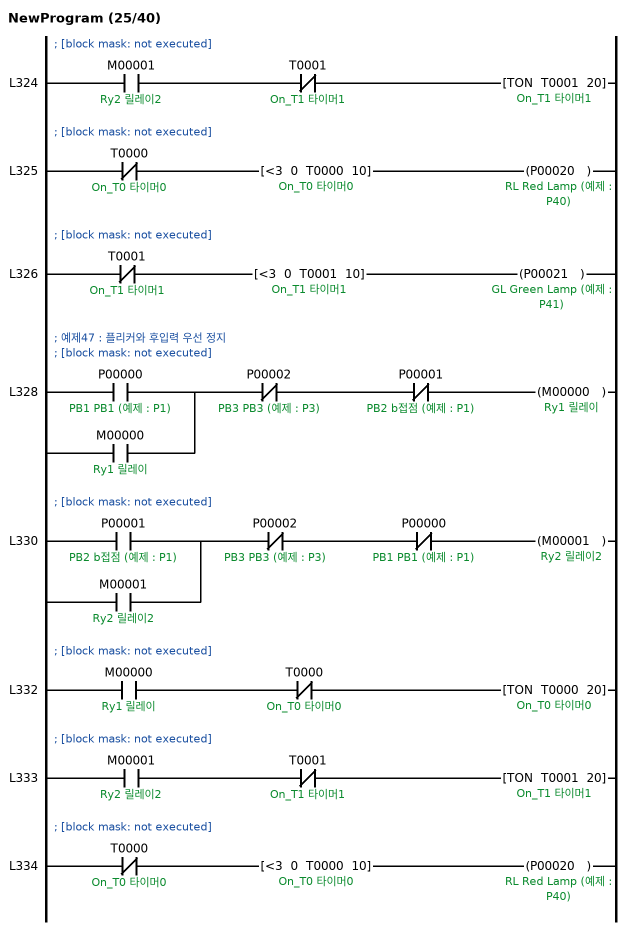
[picture p24: NewProgram rungs L324-L334]
; L324 (block mask: not executed)
LOAD      M00001	// Ry2 릴레이2
AND NOT   T0001	// On_T1 타이머1
TON       T0001 20	// On_T1 타이머1
; L325 (block mask: not executed)
LOAD NOT  T0000	// On_T0 타이머0
AND<3     0 T0000 10	// On_T0 타이머0
OUT       P00020	// RL Red Lamp (예제 : P40)
; L326 (block mask: not executed)
LOAD NOT  T0001	// On_T1 타이머1
AND<3     0 T0001 10	// On_T1 타이머1
OUT       P00021	// GL Green Lamp (예제 : P41)
// 예제47 : 플리커와 후입력 우선 정지
; L328 (block mask: not executed)
LOAD      P00000	// PB1 PB1 (예제 : P1)
OR        M00000	// Ry1 릴레이
AND NOT   P00002	// PB3 PB3 (예제 : P3)
AND NOT   P00001	// PB2 b접점 (예제 : P1)
OUT       M00000	// Ry1 릴레이
; L330 (block mask: not executed)
LOAD      P00001	// PB2 b접점 (예제 : P1)
OR        M00001	// Ry2 릴레이2
AND NOT   P00002	// PB3 PB3 (예제 : P3)
AND NOT   P00000	// PB1 PB1 (예제 : P1)
OUT       M00001	// Ry2 릴레이2
; L332 (block mask: not executed)
LOAD      M00000	// Ry1 릴레이
AND NOT   T0000	// On_T0 타이머0
TON       T0000 20	// On_T0 타이머0
; L333 (block mask: not executed)
LOAD      M00001	// Ry2 릴레이2
AND NOT   T0001	// On_T1 타이머1
TON       T0001 20	// On_T1 타이머1
; L334 (block mask: not executed)
LOAD NOT  T0000	// On_T0 타이머0
AND<3     0 T0000 10	// On_T0 타이머0
OUT       P00020	// RL Red Lamp (예제 : P40)

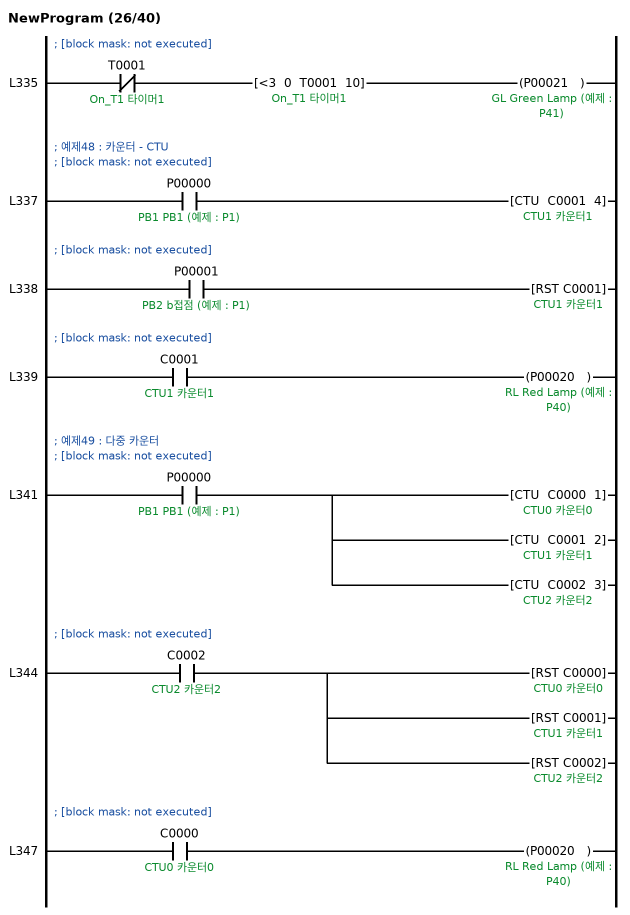
; L335 (block mask: not executed)
LOAD NOT  T0001	// On_T1 타이머1
AND<3     0 T0001 10	// On_T1 타이머1
OUT       P00021	// GL Green Lamp (예제 : P41)
// 예제48 : 카운터 - CTU
; L337 (block mask: not executed)
LOAD      P00000	// PB1 PB1 (예제 : P1)
CTU       C0001 4	// CTU1 카운터1
; L338 (block mask: not executed)
LOAD      P00001	// PB2 b접점 (예제 : P1)
RST       C0001	// CTU1 카운터1
; L339 (block mask: not executed)
LOAD      C0001	// CTU1 카운터1
OUT       P00020	// RL Red Lamp (예제 : P40)
// 예제49 : 다중 카운터
; L341 (block mask: not executed)
LOAD      P00000	// PB1 PB1 (예제 : P1)
CTU       C0000 1	// CTU0 카운터0
CTU       C0001 2	// CTU1 카운터1
CTU       C0002 3	// CTU2 카운터2
; L344 (block mask: not executed)
LOAD      C0002	// CTU2 카운터2
RST       C0000	// CTU0 카운터0
RST       C0001	// CTU1 카운터1
RST       C0002	// CTU2 카운터2
; L347 (block mask: not executed)
LOAD      C0000	// CTU0 카운터0
OUT       P00020	// RL Red Lamp (예제 : P40)

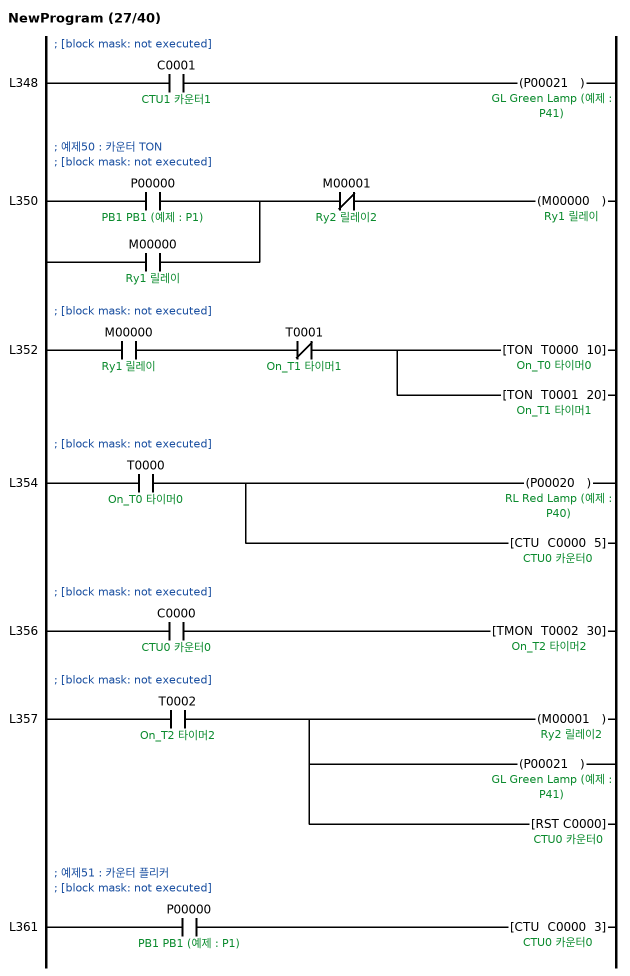
; L348 (block mask: not executed)
LOAD      C0001	// CTU1 카운터1
OUT       P00021	// GL Green Lamp (예제 : P41)
// 예제50 : 카운터 TON
; L350 (block mask: not executed)
LOAD      P00000	// PB1 PB1 (예제 : P1)
OR        M00000	// Ry1 릴레이
AND NOT   M00001	// Ry2 릴레이2
OUT       M00000	// Ry1 릴레이
; L352 (block mask: not executed)
LOAD      M00000	// Ry1 릴레이
AND NOT   T0001	// On_T1 타이머1
TON       T0000 10	// On_T0 타이머0
TON       T0001 20	// On_T1 타이머1
; L354 (block mask: not executed)
LOAD      T0000	// On_T0 타이머0
OUT       P00020	// RL Red Lamp (예제 : P40)
CTU       C0000 5	// CTU0 카운터0
; L356 (block mask: not executed)
LOAD      C0000	// CTU0 카운터0
TMON      T0002 30	// On_T2 타이머2
; L357 (block mask: not executed)
LOAD      T0002	// On_T2 타이머2
OUT       M00001	// Ry2 릴레이2
OUT       P00021	// GL Green Lamp (예제 : P41)
RST       C0000	// CTU0 카운터0
// 예제51 : 카운터 플리커
; L361 (block mask: not executed)
LOAD      P00000	// PB1 PB1 (예제 : P1)
CTU       C0000 3	// CTU0 카운터0

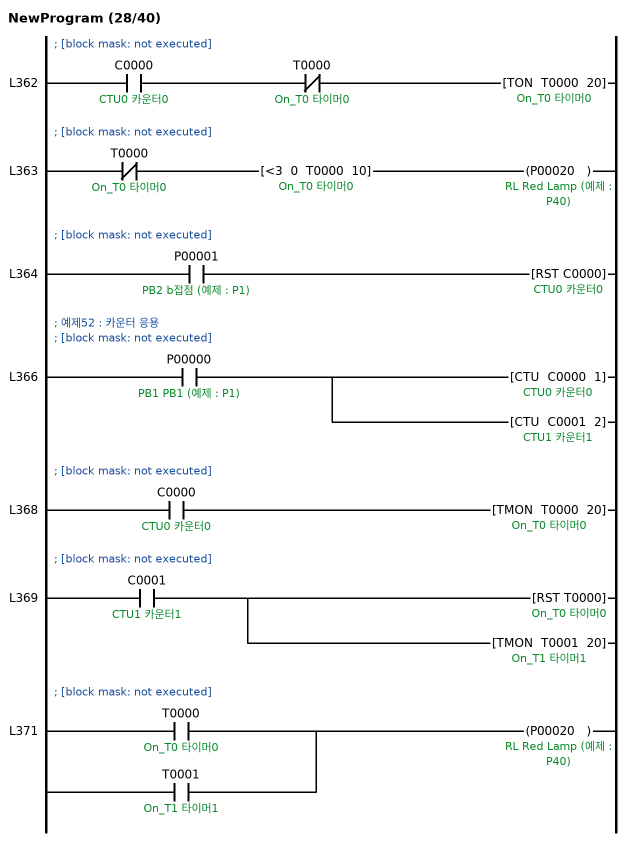
; L362 (block mask: not executed)
LOAD      C0000	// CTU0 카운터0
AND NOT   T0000	// On_T0 타이머0
TON       T0000 20	// On_T0 타이머0
; L363 (block mask: not executed)
LOAD NOT  T0000	// On_T0 타이머0
AND<3     0 T0000 10	// On_T0 타이머0
OUT       P00020	// RL Red Lamp (예제 : P40)
; L364 (block mask: not executed)
LOAD      P00001	// PB2 b접점 (예제 : P1)
RST       C0000	// CTU0 카운터0
// 예제52 : 카운터 응용
; L366 (block mask: not executed)
LOAD      P00000	// PB1 PB1 (예제 : P1)
CTU       C0000 1	// CTU0 카운터0
CTU       C0001 2	// CTU1 카운터1
; L368 (block mask: not executed)
LOAD      C0000	// CTU0 카운터0
TMON      T0000 20	// On_T0 타이머0
; L369 (block mask: not executed)
LOAD      C0001	// CTU1 카운터1
RST       T0000	// On_T0 타이머0
TMON      T0001 20	// On_T1 타이머1
; L371 (block mask: not executed)
LOAD      T0000	// On_T0 타이머0
OR        T0001	// On_T1 타이머1
OUT       P00020	// RL Red Lamp (예제 : P40)

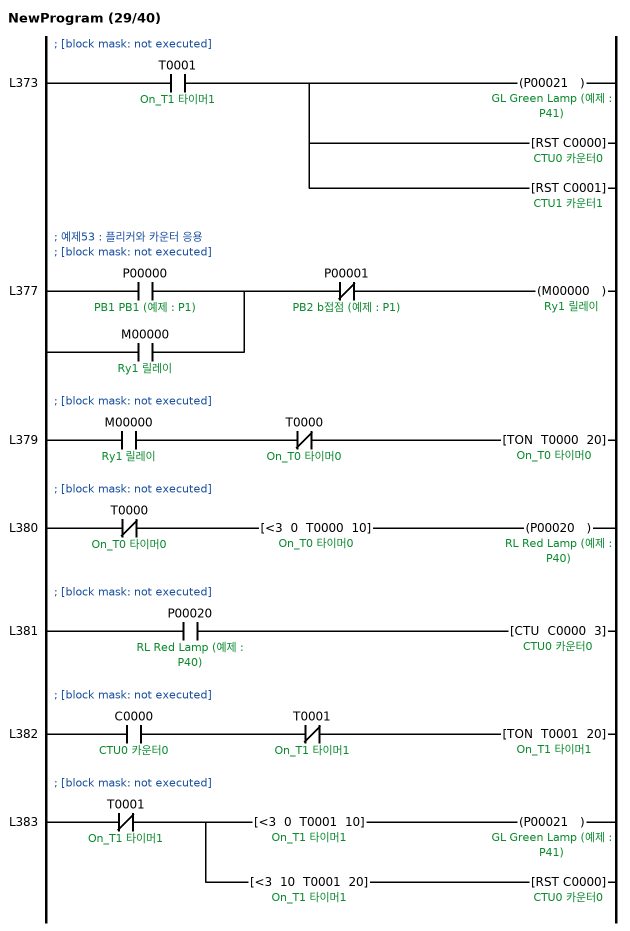
; L373 (block mask: not executed)
LOAD      T0001	// On_T1 타이머1
OUT       P00021	// GL Green Lamp (예제 : P41)
RST       C0000	// CTU0 카운터0
RST       C0001	// CTU1 카운터1
// 예제53 : 플리커와 카운터 응용
; L377 (block mask: not executed)
LOAD      P00000	// PB1 PB1 (예제 : P1)
OR        M00000	// Ry1 릴레이
AND NOT   P00001	// PB2 b접점 (예제 : P1)
OUT       M00000	// Ry1 릴레이
; L379 (block mask: not executed)
LOAD      M00000	// Ry1 릴레이
AND NOT   T0000	// On_T0 타이머0
TON       T0000 20	// On_T0 타이머0
; L380 (block mask: not executed)
LOAD NOT  T0000	// On_T0 타이머0
AND<3     0 T0000 10	// On_T0 타이머0
OUT       P00020	// RL Red Lamp (예제 : P40)
; L381 (block mask: not executed)
LOAD      P00020	// RL Red Lamp (예제 : P40)
CTU       C0000 3	// CTU0 카운터0
; L382 (block mask: not executed)
LOAD      C0000	// CTU0 카운터0
AND NOT   T0001	// On_T1 타이머1
TON       T0001 20	// On_T1 타이머1
; L383 (block mask: not executed)
LOAD NOT  T0001	// On_T1 타이머1
MPUSH
AND<3     0 T0001 10	// On_T1 타이머1
OUT       P00021	// GL Green Lamp (예제 : P41)
MPOP
AND<3     10 T0001 20	// On_T1 타이머1
RST       C0000	// CTU0 카운터0

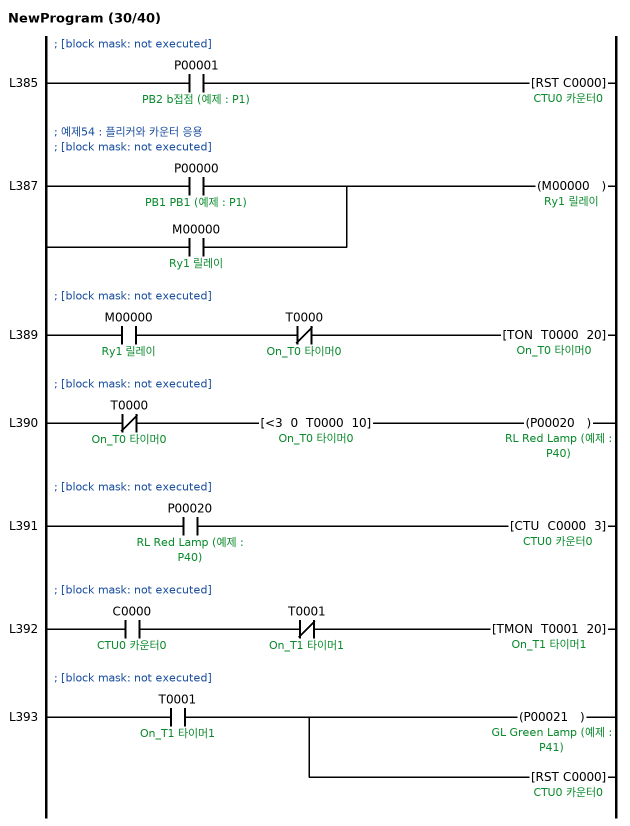
; L385 (block mask: not executed)
LOAD      P00001	// PB2 b접점 (예제 : P1)
RST       C0000	// CTU0 카운터0
// 예제54 : 플리커와 카운터 응용
; L387 (block mask: not executed)
LOAD      P00000	// PB1 PB1 (예제 : P1)
OR        M00000	// Ry1 릴레이
OUT       M00000	// Ry1 릴레이
; L389 (block mask: not executed)
LOAD      M00000	// Ry1 릴레이
AND NOT   T0000	// On_T0 타이머0
TON       T0000 20	// On_T0 타이머0
; L390 (block mask: not executed)
LOAD NOT  T0000	// On_T0 타이머0
AND<3     0 T0000 10	// On_T0 타이머0
OUT       P00020	// RL Red Lamp (예제 : P40)
; L391 (block mask: not executed)
LOAD      P00020	// RL Red Lamp (예제 : P40)
CTU       C0000 3	// CTU0 카운터0
; L392 (block mask: not executed)
LOAD      C0000	// CTU0 카운터0
AND NOT   T0001	// On_T1 타이머1
TMON      T0001 20	// On_T1 타이머1
; L393 (block mask: not executed)
LOAD      T0001	// On_T1 타이머1
OUT       P00021	// GL Green Lamp (예제 : P41)
RST       C0000	// CTU0 카운터0

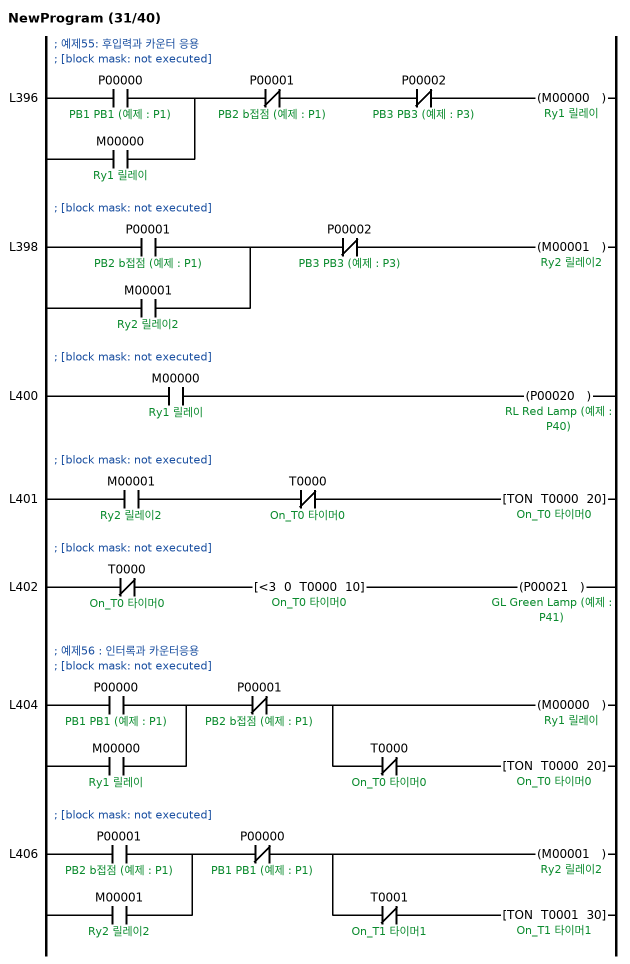
// 예제55: 후입력과 카운터 응용
; L396 (block mask: not executed)
LOAD      P00000	// PB1 PB1 (예제 : P1)
OR        M00000	// Ry1 릴레이
AND NOT   P00001	// PB2 b접점 (예제 : P1)
AND NOT   P00002	// PB3 PB3 (예제 : P3)
OUT       M00000	// Ry1 릴레이
; L398 (block mask: not executed)
LOAD      P00001	// PB2 b접점 (예제 : P1)
OR        M00001	// Ry2 릴레이2
AND NOT   P00002	// PB3 PB3 (예제 : P3)
OUT       M00001	// Ry2 릴레이2
; L400 (block mask: not executed)
LOAD      M00000	// Ry1 릴레이
OUT       P00020	// RL Red Lamp (예제 : P40)
; L401 (block mask: not executed)
LOAD      M00001	// Ry2 릴레이2
AND NOT   T0000	// On_T0 타이머0
TON       T0000 20	// On_T0 타이머0
; L402 (block mask: not executed)
LOAD NOT  T0000	// On_T0 타이머0
AND<3     0 T0000 10	// On_T0 타이머0
OUT       P00021	// GL Green Lamp (예제 : P41)
// 예제56 : 인터록과 카운터응용
; L404 (block mask: not executed)
LOAD      P00000	// PB1 PB1 (예제 : P1)
OR        M00000	// Ry1 릴레이
AND NOT   P00001	// PB2 b접점 (예제 : P1)
OUT       M00000	// Ry1 릴레이
AND NOT   T0000	// On_T0 타이머0
TON       T0000 20	// On_T0 타이머0
; L406 (block mask: not executed)
LOAD      P00001	// PB2 b접점 (예제 : P1)
OR        M00001	// Ry2 릴레이2
AND NOT   P00000	// PB1 PB1 (예제 : P1)
OUT       M00001	// Ry2 릴레이2
AND NOT   T0001	// On_T1 타이머1
TON       T0001 30	// On_T1 타이머1

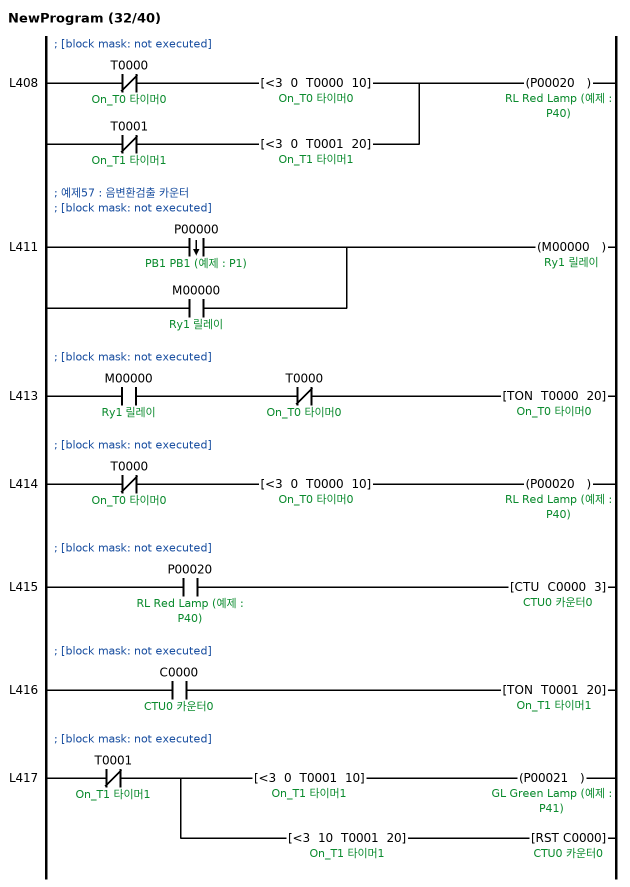
; L408 (block mask: not executed)
LOAD NOT  T0000	// On_T0 타이머0
AND<3     0 T0000 10	// On_T0 타이머0
LOAD NOT  T0001	// On_T1 타이머1
AND<3     0 T0001 20	// On_T1 타이머1
OR LOAD
OUT       P00020	// RL Red Lamp (예제 : P40)
// 예제57 : 음변환검출 카운터
; L411 (block mask: not executed)
LOADN     P00000	// PB1 PB1 (예제 : P1)
OR        M00000	// Ry1 릴레이
OUT       M00000	// Ry1 릴레이
; L413 (block mask: not executed)
LOAD      M00000	// Ry1 릴레이
AND NOT   T0000	// On_T0 타이머0
TON       T0000 20	// On_T0 타이머0
; L414 (block mask: not executed)
LOAD NOT  T0000	// On_T0 타이머0
AND<3     0 T0000 10	// On_T0 타이머0
OUT       P00020	// RL Red Lamp (예제 : P40)
; L415 (block mask: not executed)
LOAD      P00020	// RL Red Lamp (예제 : P40)
CTU       C0000 3	// CTU0 카운터0
; L416 (block mask: not executed)
LOAD      C0000	// CTU0 카운터0
TON       T0001 20	// On_T1 타이머1
; L417 (block mask: not executed)
LOAD NOT  T0001	// On_T1 타이머1
MPUSH
AND<3     0 T0001 10	// On_T1 타이머1
OUT       P00021	// GL Green Lamp (예제 : P41)
MPOP
AND<3     10 T0001 20	// On_T1 타이머1
RST       C0000	// CTU0 카운터0

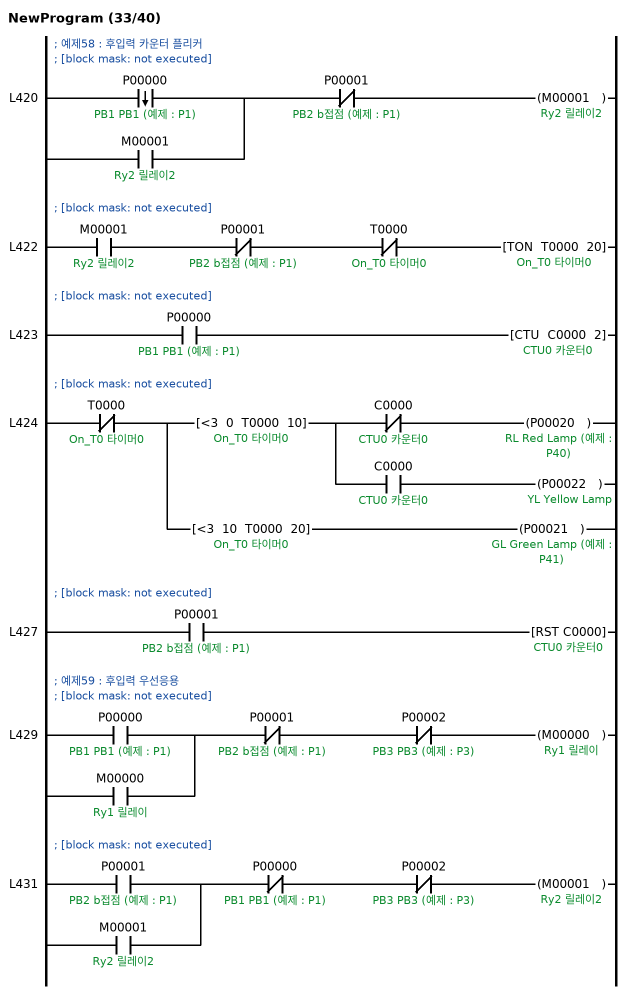
// 예제58 : 후입력 카운터 플리커
; L420 (block mask: not executed)
LOADN     P00000	// PB1 PB1 (예제 : P1)
OR        M00001	// Ry2 릴레이2
AND NOT   P00001	// PB2 b접점 (예제 : P1)
OUT       M00001	// Ry2 릴레이2
; L422 (block mask: not executed)
LOAD      M00001	// Ry2 릴레이2
AND NOT   P00001	// PB2 b접점 (예제 : P1)
AND NOT   T0000	// On_T0 타이머0
TON       T0000 20	// On_T0 타이머0
; L423 (block mask: not executed)
LOAD      P00000	// PB1 PB1 (예제 : P1)
CTU       C0000 2	// CTU0 카운터0
; L424 (block mask: not executed)
LOAD NOT  T0000	// On_T0 타이머0
MPUSH
AND<3     0 T0000 10	// On_T0 타이머0
MPUSH
AND NOT   C0000	// CTU0 카운터0
OUT       P00020	// RL Red Lamp (예제 : P40)
MPOP
AND       C0000	// CTU0 카운터0
OUT       P00022	// YL Yellow Lamp
MPOP
AND<3     10 T0000 20	// On_T0 타이머0
OUT       P00021	// GL Green Lamp (예제 : P41)
; L427 (block mask: not executed)
LOAD      P00001	// PB2 b접점 (예제 : P1)
RST       C0000	// CTU0 카운터0
// 예제59 : 후입력 우선응용
; L429 (block mask: not executed)
LOAD      P00000	// PB1 PB1 (예제 : P1)
OR        M00000	// Ry1 릴레이
AND NOT   P00001	// PB2 b접점 (예제 : P1)
AND NOT   P00002	// PB3 PB3 (예제 : P3)
OUT       M00000	// Ry1 릴레이
; L431 (block mask: not executed)
LOAD      P00001	// PB2 b접점 (예제 : P1)
OR        M00001	// Ry2 릴레이2
AND NOT   P00000	// PB1 PB1 (예제 : P1)
AND NOT   P00002	// PB3 PB3 (예제 : P3)
OUT       M00001	// Ry2 릴레이2

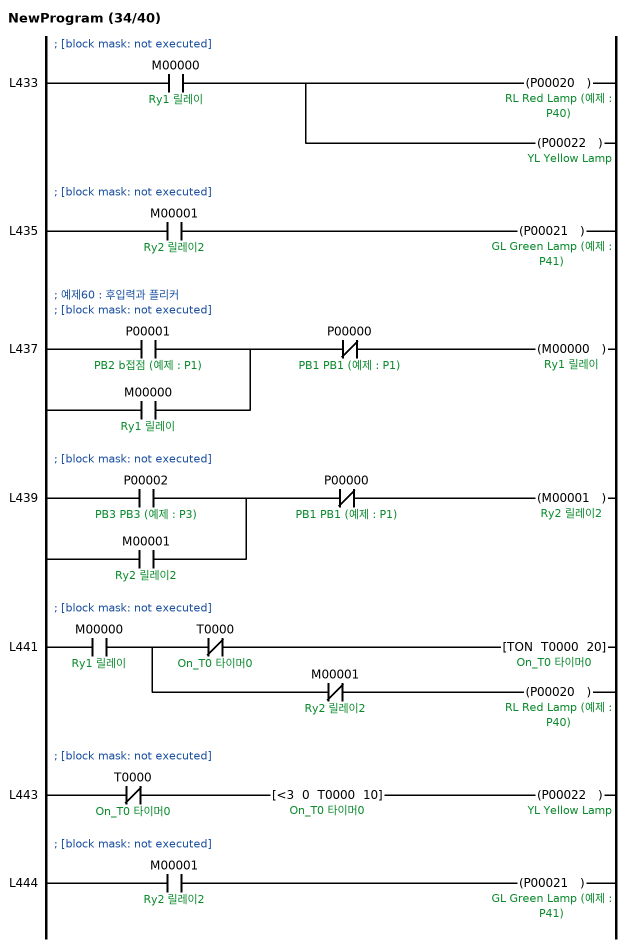
; L433 (block mask: not executed)
LOAD      M00000	// Ry1 릴레이
OUT       P00020	// RL Red Lamp (예제 : P40)
OUT       P00022	// YL Yellow Lamp
; L435 (block mask: not executed)
LOAD      M00001	// Ry2 릴레이2
OUT       P00021	// GL Green Lamp (예제 : P41)
// 예제60 : 후입력과 플리커
; L437 (block mask: not executed)
LOAD      P00001	// PB2 b접점 (예제 : P1)
OR        M00000	// Ry1 릴레이
AND NOT   P00000	// PB1 PB1 (예제 : P1)
OUT       M00000	// Ry1 릴레이
; L439 (block mask: not executed)
LOAD      P00002	// PB3 PB3 (예제 : P3)
OR        M00001	// Ry2 릴레이2
AND NOT   P00000	// PB1 PB1 (예제 : P1)
OUT       M00001	// Ry2 릴레이2
; L441 (block mask: not executed)
LOAD      M00000	// Ry1 릴레이
MPUSH
AND NOT   T0000	// On_T0 타이머0
TON       T0000 20	// On_T0 타이머0
MPOP
AND NOT   M00001	// Ry2 릴레이2
OUT       P00020	// RL Red Lamp (예제 : P40)
; L443 (block mask: not executed)
LOAD NOT  T0000	// On_T0 타이머0
AND<3     0 T0000 10	// On_T0 타이머0
OUT       P00022	// YL Yellow Lamp
; L444 (block mask: not executed)
LOAD      M00001	// Ry2 릴레이2
OUT       P00021	// GL Green Lamp (예제 : P41)

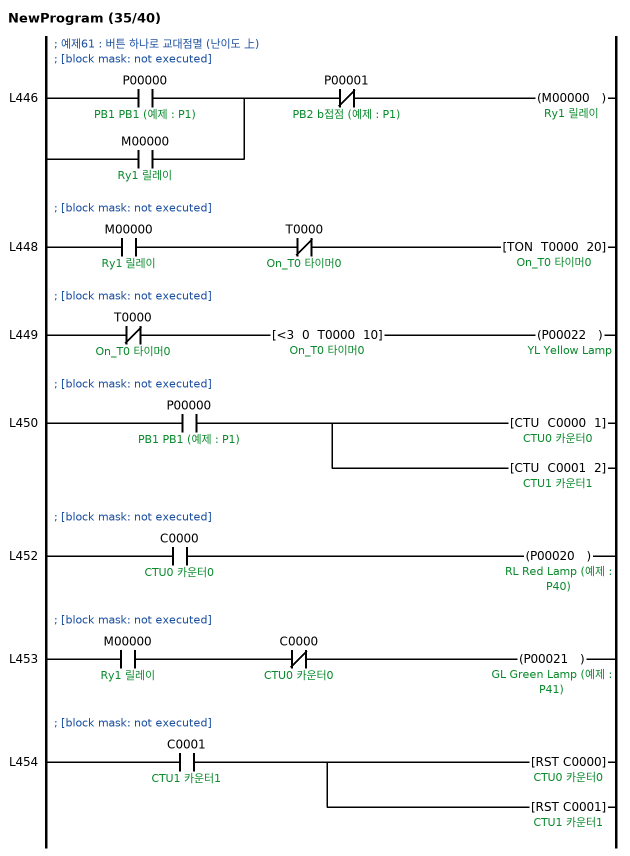
// 예제61 : 버튼 하나로 교대점멸 (난이도 上)
; L446 (block mask: not executed)
LOAD      P00000	// PB1 PB1 (예제 : P1)
OR        M00000	// Ry1 릴레이
AND NOT   P00001	// PB2 b접점 (예제 : P1)
OUT       M00000	// Ry1 릴레이
; L448 (block mask: not executed)
LOAD      M00000	// Ry1 릴레이
AND NOT   T0000	// On_T0 타이머0
TON       T0000 20	// On_T0 타이머0
; L449 (block mask: not executed)
LOAD NOT  T0000	// On_T0 타이머0
AND<3     0 T0000 10	// On_T0 타이머0
OUT       P00022	// YL Yellow Lamp
; L450 (block mask: not executed)
LOAD      P00000	// PB1 PB1 (예제 : P1)
CTU       C0000 1	// CTU0 카운터0
CTU       C0001 2	// CTU1 카운터1
; L452 (block mask: not executed)
LOAD      C0000	// CTU0 카운터0
OUT       P00020	// RL Red Lamp (예제 : P40)
; L453 (block mask: not executed)
LOAD      M00000	// Ry1 릴레이
AND NOT   C0000	// CTU0 카운터0
OUT       P00021	// GL Green Lamp (예제 : P41)
; L454 (block mask: not executed)
LOAD      C0001	// CTU1 카운터1
RST       C0000	// CTU0 카운터0
RST       C0001	// CTU1 카운터1

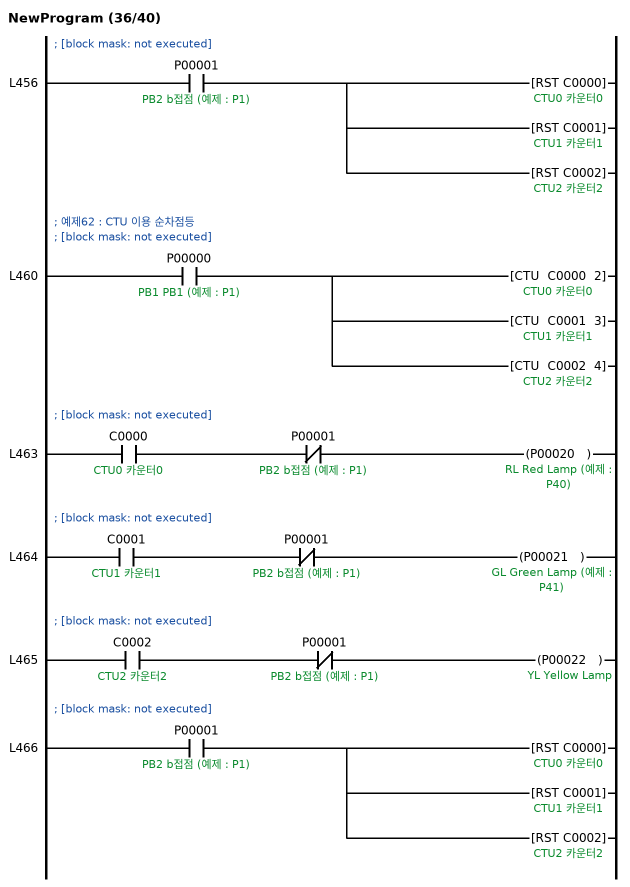
; L456 (block mask: not executed)
LOAD      P00001	// PB2 b접점 (예제 : P1)
RST       C0000	// CTU0 카운터0
RST       C0001	// CTU1 카운터1
RST       C0002	// CTU2 카운터2
// 예제62 : CTU 이용 순차점등
; L460 (block mask: not executed)
LOAD      P00000	// PB1 PB1 (예제 : P1)
CTU       C0000 2	// CTU0 카운터0
CTU       C0001 3	// CTU1 카운터1
CTU       C0002 4	// CTU2 카운터2
; L463 (block mask: not executed)
LOAD      C0000	// CTU0 카운터0
AND NOT   P00001	// PB2 b접점 (예제 : P1)
OUT       P00020	// RL Red Lamp (예제 : P40)
; L464 (block mask: not executed)
LOAD      C0001	// CTU1 카운터1
AND NOT   P00001	// PB2 b접점 (예제 : P1)
OUT       P00021	// GL Green Lamp (예제 : P41)
; L465 (block mask: not executed)
LOAD      C0002	// CTU2 카운터2
AND NOT   P00001	// PB2 b접점 (예제 : P1)
OUT       P00022	// YL Yellow Lamp
; L466 (block mask: not executed)
LOAD      P00001	// PB2 b접점 (예제 : P1)
RST       C0000	// CTU0 카운터0
RST       C0001	// CTU1 카운터1
RST       C0002	// CTU2 카운터2

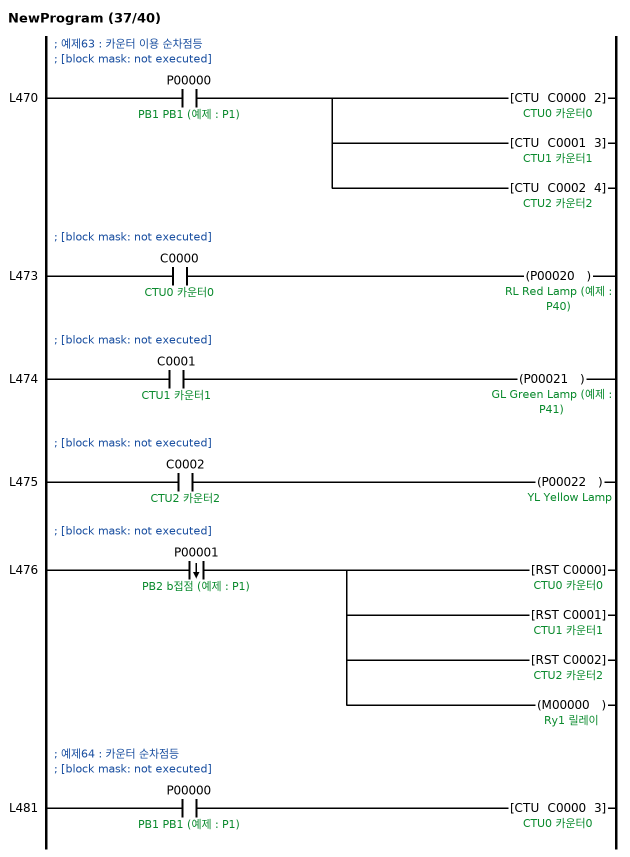
// 예제63 : 카운터 이용 순차점등
; L470 (block mask: not executed)
LOAD      P00000	// PB1 PB1 (예제 : P1)
CTU       C0000 2	// CTU0 카운터0
CTU       C0001 3	// CTU1 카운터1
CTU       C0002 4	// CTU2 카운터2
; L473 (block mask: not executed)
LOAD      C0000	// CTU0 카운터0
OUT       P00020	// RL Red Lamp (예제 : P40)
; L474 (block mask: not executed)
LOAD      C0001	// CTU1 카운터1
OUT       P00021	// GL Green Lamp (예제 : P41)
; L475 (block mask: not executed)
LOAD      C0002	// CTU2 카운터2
OUT       P00022	// YL Yellow Lamp
; L476 (block mask: not executed)
LOADN     P00001	// PB2 b접점 (예제 : P1)
RST       C0000	// CTU0 카운터0
RST       C0001	// CTU1 카운터1
RST       C0002	// CTU2 카운터2
OUT       M00000	// Ry1 릴레이
// 예제64 : 카운터 순차점등
; L481 (block mask: not executed)
LOAD      P00000	// PB1 PB1 (예제 : P1)
CTU       C0000 3	// CTU0 카운터0

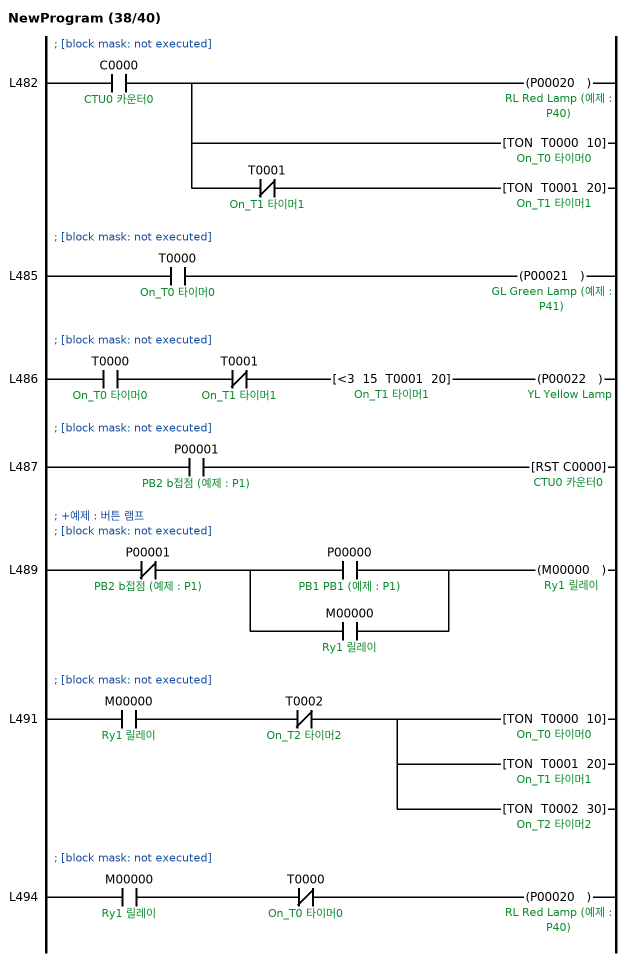
; L482 (block mask: not executed)
LOAD      C0000	// CTU0 카운터0
OUT       P00020	// RL Red Lamp (예제 : P40)
TON       T0000 10	// On_T0 타이머0
AND NOT   T0001	// On_T1 타이머1
TON       T0001 20	// On_T1 타이머1
; L485 (block mask: not executed)
LOAD      T0000	// On_T0 타이머0
OUT       P00021	// GL Green Lamp (예제 : P41)
; L486 (block mask: not executed)
LOAD      T0000	// On_T0 타이머0
AND NOT   T0001	// On_T1 타이머1
AND<3     15 T0001 20	// On_T1 타이머1
OUT       P00022	// YL Yellow Lamp
; L487 (block mask: not executed)
LOAD      P00001	// PB2 b접점 (예제 : P1)
RST       C0000	// CTU0 카운터0
// +예제 : 버튼 램프
; L489 (block mask: not executed)
LOAD NOT  P00001	// PB2 b접점 (예제 : P1)
LOAD      P00000	// PB1 PB1 (예제 : P1)
OR        M00000	// Ry1 릴레이
AND LOAD
OUT       M00000	// Ry1 릴레이
; L491 (block mask: not executed)
LOAD      M00000	// Ry1 릴레이
AND NOT   T0002	// On_T2 타이머2
TON       T0000 10	// On_T0 타이머0
TON       T0001 20	// On_T1 타이머1
TON       T0002 30	// On_T2 타이머2
; L494 (block mask: not executed)
LOAD      M00000	// Ry1 릴레이
AND NOT   T0000	// On_T0 타이머0
OUT       P00020	// RL Red Lamp (예제 : P40)

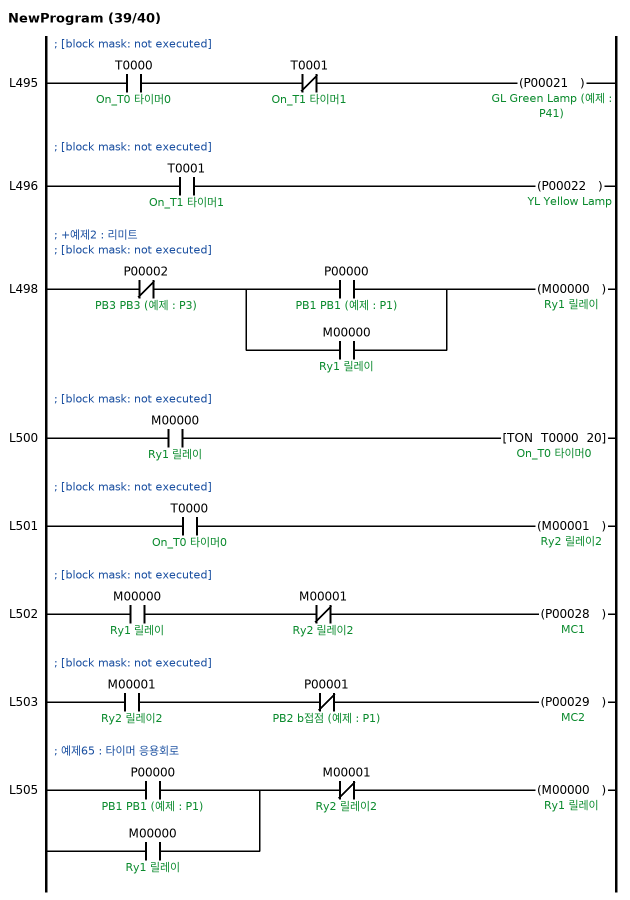
; L495 (block mask: not executed)
LOAD      T0000	// On_T0 타이머0
AND NOT   T0001	// On_T1 타이머1
OUT       P00021	// GL Green Lamp (예제 : P41)
; L496 (block mask: not executed)
LOAD      T0001	// On_T1 타이머1
OUT       P00022	// YL Yellow Lamp
// +예제2 : 리미트
; L498 (block mask: not executed)
LOAD NOT  P00002	// PB3 PB3 (예제 : P3)
LOAD      P00000	// PB1 PB1 (예제 : P1)
OR        M00000	// Ry1 릴레이
AND LOAD
OUT       M00000	// Ry1 릴레이
; L500 (block mask: not executed)
LOAD      M00000	// Ry1 릴레이
TON       T0000 20	// On_T0 타이머0
; L501 (block mask: not executed)
LOAD      T0000	// On_T0 타이머0
OUT       M00001	// Ry2 릴레이2
; L502 (block mask: not executed)
LOAD      M00000	// Ry1 릴레이
AND NOT   M00001	// Ry2 릴레이2
OUT       P00028	// MC1
; L503 (block mask: not executed)
LOAD      M00001	// Ry2 릴레이2
AND NOT   P00001	// PB2 b접점 (예제 : P1)
OUT       P00029	// MC2
// 예제65 : 타이머 응용회로
; L505
LOAD      P00000	// PB1 PB1 (예제 : P1)
OR        M00000	// Ry1 릴레이
AND NOT   M00001	// Ry2 릴레이2
OUT       M00000	// Ry1 릴레이

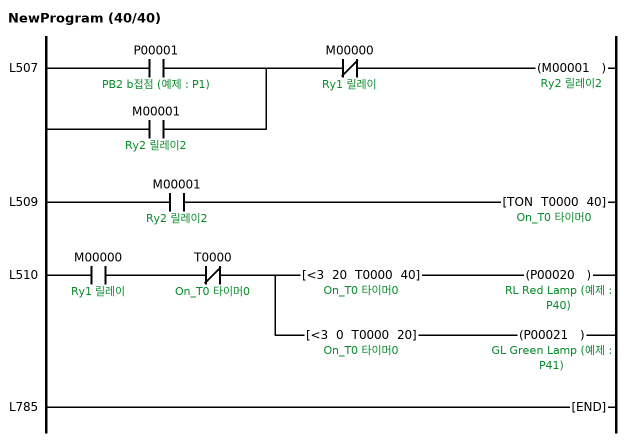
; L507
LOAD      P00001	// PB2 b접점 (예제 : P1)
OR        M00001	// Ry2 릴레이2
AND NOT   M00000	// Ry1 릴레이
OUT       M00001	// Ry2 릴레이2
; L509
LOAD      M00001	// Ry2 릴레이2
TON       T0000 40	// On_T0 타이머0
; L510
LOAD      M00000	// Ry1 릴레이
AND NOT   T0000	// On_T0 타이머0
MPUSH
AND<3     20 T0000 40	// On_T0 타이머0
OUT       P00020	// RL Red Lamp (예제 : P40)
MPOP
AND<3     0 T0000 20	// On_T0 타이머0
OUT       P00021	// GL Green Lamp (예제 : P41)
; L785
END

VARIABLES AND COMMENTS (devices not used above)
P00031	BIT	MC2
P00030	BIT	MC1